// TIA Portal project "AWL LIBRO 3" (V11)

(* hardware
DEVICE "S7300/ET200 station_1"  SIMATIC 300-Station
   slot 0: "Perfil soporte_0"  Rail  6ES7 390-1***0-0AA0
   slot 2: "PLC_1"  CPU 313C-2 DP  6ES7 313-6CF03-0AB0  V2.6
      slot 0: "Interfaz MPI_1"  MPI
      slot 1: "Interfaz DP_1"  DP
      slot 2: "DI16/DO16_1"  DI16/DO16
      slot 4: "Contaje_1"  Counter
*)

// ===== PLC "PLC_1"  CPU 313C-2 DP =====

VAR_GLOBAL   // PLC tag table "Tabla de variables estándar"
   "PARO." AT %E0.0 : Bool;
   "MARCHA." AT %E0.1 : Bool;
   "FINAL DE CARRERA" AT %E0.2 : Bool;
   "CELULA FOTOELCTRICA" AT %E0.3 : Bool;
   "C. TRANSPORTADORA" AT %A0.0 : Bool;
   "MOTOR TALADRO" AT %A0.1 : Bool;
   "PISTON RECOGIDO" AT %A0.2 : Bool;
   "PISTON EXPANDIDO" AT %A0.3 : Bool;
   "Tag_1" AT %M10.0 : Bool;
   "SALIDAS" AT %AB0 : Byte;
   "Tag_2" AT %M10.1 : Bool;
   "Tag_3" AT %M30.0 : Bool;
   "Tag_4" AT %T0 : Timer;
   "Tag_5" AT %M10.2 : Bool;
   "Tag_7" AT %T1 : Timer;
   "Tag_8" AT %M10.3 : Bool;
   "LED PARO" AT %A0.4 : Bool;
END_VAR

ORGANIZATION_BLOCK "Main"   // OB1, STL
TITLE = EJERCICIO 3 LIBRO / "Main Program Sweep (Cycle)"
{ S7_Optimized_Access := 'FALSE' }
VERSION : 0.1
   VAR_TEMP
      OB1_EV_CLASS : Byte;   // Bits 0-3 = 1 (Coming event), Bits 4-7 = 1 (Event class 1)
      OB1_SCAN_1 : Byte;   // 1 (Cold restart scan 1 of OB 1), 3 (Scan 2-n of OB 1)
      OB1_PRIORITY : Byte;   // Priority of OB Execution
      OB1_OB_NUMBR : Byte;   // 1 (Organization block 1, OB1)
      OB1_RESERVED_1 : Byte;   // Reserved for system
      OB1_RESERVED_2 : Byte;   // Reserved for system
      OB1_PREV_CYCLE : Int;   // Cycle time of previous OB1 scan (milliseconds)
      OB1_MIN_CYCLE : Int;   // Minimum cycle time of OB1 (milliseconds)
      OB1_MAX_CYCLE : Int;   // Maximum cycle time of OB1 (milliseconds)
      OB1_DATE_TIME : Date_And_Time;   // Date and time OB1 started
   END_VAR
BEGIN

REGION Network 1
         A     "PARO.";  // PARO REPOSO.
         FP    "Tag_8";
         JNB   _004;
         L     B#16#10;
         T     "SALIDAS";
   _004: NOP   0;
         NOP   0;
         O     "MARCHA.";  // INICIO PROCESO.
         O     "PISTON RECOGIDO";
         A     "FINAL DE CARRERA";  // TIENE QUE ESTAR PRESIONADO PARA INICIAR LA MARCHA.
         FP    "Tag_1";
         JNB   _001;
         L     B#16#07;
         T     "SALIDAS";
   _001: NOP   0;
         A     "CELULA FOTOELCTRICA";  // DETECCION CELULA FOTOELECTRICA.
         FP    "Tag_2";
         S     "Tag_3";  // SET BOBINA AUXILIAR ALIENTACION T0.
         A     "Tag_3";
         L     S5T#2S;  // TEMPORIZADO 2S.
         SD    "Tag_4";
         O     "Tag_4";  // CONTACTO T0.
         O     "Tag_7";

         FP    "Tag_5";
         JNB   _002;
         L     B#16#6;
         T     "SALIDAS";
         R     "Tag_3";
   _002: NOP   0;
         A     "Tag_4";  // ACTIVACION VAVULA.
         JNB   _003;
         L     B#16#A;
         T     "SALIDAS";
   _003: NOP   0;
         A     "PISTON EXPANDIDO";  // PERFORACION PIEZA.
         L     S5T#3S;
         SD    "Tag_7";
END_REGION
END_ORGANIZATION_BLOCK